TYPE ST_System_Ampel_Stellwert :
STRUCT
	Stellung_Rot		: BOOL;
	Stellung_Orange		: BOOL;
	Stellung_Gruen		: BOOL;
	Stellung_Blau		: BOOL;
	Stellung_Buzz		: BOOL;
END_STRUCT
END_TYPE

(* stored: Version 1.1.0.1, ProductVersion 3.1.4024.9
   DUT ST_System_Ampel_Stellwert: Id {0f7e4c6c-c502-45fd-9b89-a22851b7756f} *)
